Omron Sysmac Studio project SPA_P3 (Sysmac Studio 1.23.0.14, StandardProject)

# Controller new_Controller_0: NX1P2-1040DT1 version 1.18
Task PrimaryTask (priority 4, period or condition 2000): Programa0

PROGRAM Programa0
VAR
    weight : REAL;
    frequency : REAL;
    limitedWeight : REAL;
END_VAR

(* Section MAIN: ladder, written here as Structured Text *)

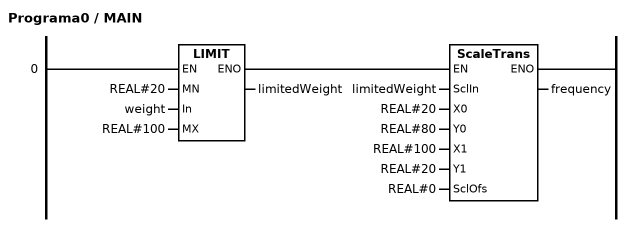
(* Rung 0 *)
limitedWeight := LIMIT(MN := REAL#20, In := weight, MX := REAL#100);
frequency := ScaleTrans(SclIn := limitedWeight, X0 := REAL#20, Y0 := REAL#80, X1 := REAL#100, Y1 := REAL#20, SclOfs := REAL#0);
END_PROGRAM